// TIA Portal V20 export
DATA_BLOCK "IDB_Flow_Test"   // DB46
// stored: InstanceOfName ProductionLine.Flow_Test, InstanceOfType FB, Namespace ProductionLine
"ProductionLine.Flow_Test"
   // VAR
   //    Start { S7_SetPoint := 'True'} : Bool;
   //    StartTest { S7_SetPoint := 'True'} : "ProductionLine.Test_Logic";
   //    GoToRightDP1 { S7_SetPoint := 'True'} : "ProductionLine.Test_Logic";
   //    ContinueStraightDP1 { S7_SetPoint := 'True'} : "ProductionLine.Test_Logic";
   //    ContinueStraightDP2 { S7_SetPoint := 'True'} : "ProductionLine.Test_Logic";
   //    GotorightDP2Thentoright { S7_SetPoint := 'True'} : "ProductionLine.Test_Logic";
   //    GotorightDP2ThentoLeft { S7_SetPoint := 'True'} : "ProductionLine.Test_Logic";
   //    ContinueStraightDP3 { S7_SetPoint := 'True'} : "ProductionLine.Test_Logic";
   //    ContinueStraightDP4 { S7_SetPoint := 'True'} : "ProductionLine.Test_Logic";
   //    GotoRightDP4 { S7_SetPoint := 'True'} : "ProductionLine.Test_Logic";
   //    "A1.13.1_Straight" { S7_SetPoint := 'True'} : "ProductionLine.Test_Logic";
   //    "A1.13.1_left" { S7_SetPoint := 'True'} : "ProductionLine.Test_Logic";
   //    R_TRIG_Instance { S7_SetPoint := 'True'} : R_TRIG;
   // END_VAR
BEGIN
END_DATA_BLOCK
